KUKA KRL program: Makrosaw.src

&ACCESS RV
&PARAM TPVW_VERSION=3.3.5
DEF  MAKROSAW ( )
; FOLD Makro Anfang;%{SE} %MKUKATPVW
SPS_N=-1
VW (#VW_INIT,FALSE)
SPS_N=-1
; ENDFOLD
; FOLD ;%{H}
END
; ENDFOLD
